FUNCTION_BLOCK FB_SimulatedProcessEquipment IMPLEMENTS I_ProcessEquipment
VAR
    eState : E_ProcessEquipmentState := E_ProcessEquipmentState.Ready;
    stResult : ST_ProcessResult;
    tonProcess : TON;
    bStartPending : BOOL;
    bForcePass : BOOL := TRUE;
    bForceFault : BOOL;
END_VAR

METHOD PUBLIC Cyclic
CASE eState OF
E_ProcessEquipmentState.Ready:
    IF bStartPending THEN bStartPending := FALSE; stResult.bValid := FALSE; eState := E_ProcessEquipmentState.Busy; END_IF
E_ProcessEquipmentState.Busy:
    tonProcess(IN := TRUE, PT := T#2S);
    IF bForceFault THEN eState := E_ProcessEquipmentState.Fault;
    ELSIF tonProcess.Q THEN
        tonProcess(IN := FALSE);
        stResult.bValid := TRUE; stResult.bPassed := bForcePass;
        IF bForcePass THEN stResult.eCode := E_ProcessResultCode.Pass; ELSE stResult.eCode := E_ProcessResultCode.Fail; END_IF
        stResult.sDetail := 'Simulated silicone process result';
        eState := E_ProcessEquipmentState.Completed;
    END_IF
E_ProcessEquipmentState.Completed: ;
E_ProcessEquipmentState.Fault: ;
END_CASE
END_METHOD

METHOD PUBLIC GetResult : ST_ProcessResult
GetResult := stResult;
END_METHOD

METHOD PUBLIC GetState : E_ProcessEquipmentState
GetState := eState;
END_METHOD

METHOD PUBLIC IsBusy : BOOL
IsBusy := eState = E_ProcessEquipmentState.Busy;
END_METHOD

METHOD PUBLIC IsDone : BOOL
IsDone := eState = E_ProcessEquipmentState.Completed;
END_METHOD

METHOD PUBLIC IsFaulted : BOOL
IsFaulted := eState = E_ProcessEquipmentState.Fault;
END_METHOD

METHOD PUBLIC IsReady : BOOL
IsReady := eState = E_ProcessEquipmentState.Ready;
END_METHOD

METHOD PUBLIC RequestReset
bForceFault := FALSE; stResult.bValid := FALSE; eState := E_ProcessEquipmentState.Ready;
END_METHOD

METHOD PUBLIC RequestStart : BOOL
IF eState = E_ProcessEquipmentState.Ready THEN bStartPending := TRUE; RequestStart := TRUE; END_IF
END_METHOD

METHOD PUBLIC RequestStop
bStartPending := FALSE; tonProcess(IN := FALSE); eState := E_ProcessEquipmentState.Ready;
END_METHOD

METHOD PUBLIC SetRecipe : BOOL
VAR_INPUT usiRecipe : USINT; END_VAR
stResult.usiRecipe := usiRecipe; SetRecipe := TRUE;
END_METHOD

METHOD PUBLIC SetSimulationResult
VAR_INPUT bPass : BOOL; bFault : BOOL; END_VAR
bForcePass := bPass; bForceFault := bFault;
END_METHOD

END_FUNCTION_BLOCK

(* stored: Version 1.1.0.1, ProductVersion 3.1.4026.18
   POU FB_SimulatedProcessEquipment: Id {c73d2e61-13e5-49d3-9472-ef88ed21cc93}, SpecialFunc None
   Method Cyclic: Id {3d89a91f-d8dd-4ac4-8fca-5735d3b47a29}
   Method GetResult: Id {8b4228d5-23b0-4ebf-aea9-cdf926af415c}
   Method GetState: Id {0ac6846f-e961-4778-b458-42a285c55751}
   Method IsBusy: Id {5a13f073-7ce0-49bc-9ebf-8dc4899ad23d}
   Method IsDone: Id {ef1ae204-e0a9-42bf-b4a5-1dbbba34b97c}
   Method IsFaulted: Id {21a3e40a-a951-46f5-8ee0-f7cd74f7fd4c}
   Method IsReady: Id {ad960a28-5048-49d7-a298-d3d0751caf0f}
   Method RequestReset: Id {cb5d5bfa-434e-41c2-b66e-2a4f6fb92a29}
   Method RequestStart: Id {9a67b0a8-a4c5-442a-8334-305fa330e01f}
   Method RequestStop: Id {e46c98cf-541e-44ca-b173-a79a66c20042}
   Method SetRecipe: Id {f7145259-8bd9-45fb-a7ad-40d0a3b804d9}
   Method SetSimulationResult: Id {5a1b7d3f-eaf2-481a-b1ba-b528770787e9} *)
